FUNCTION_BLOCK CALIBRATE_3P (* 3-point calibration for joysticks (Min, Mid, Max) *)
  (* Standard: 61499-1; Description: Calibrate_3P allows for 3-point calibration of an analog input, ideal for joysticks with center drift. *)
  (* Version 1.0, 2026-05-10, Gemini CLI *)
  PACKAGE OSCAT::Basic::POUs::Engineering::measurements;
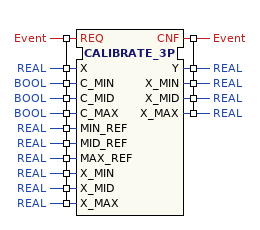
  EVENT_INPUT
    REQ WITH X, C_MIN, C_MID, C_MAX, MIN_REF, MID_REF, MAX_REF, X_MIN, X_MID, X_MAX; (* Normal Execution Request *)
  END_EVENT
  EVENT_OUTPUT
    CNF WITH Y, X_MIN, X_MID, X_MAX; (* Execution Confirmation *)
  END_EVENT
  VAR_INPUT
    X : REAL; (* Raw Input *)
    C_MIN : BOOL; (* Calibrate Min Point *)
    C_MID : BOOL; (* Calibrate Mid Point (Center) *)
    C_MAX : BOOL; (* Calibrate Max Point *)
    MIN_REF : REAL := 0.0; (* Target value for Min *)
    MID_REF : REAL := 50.0; (* Target value for Mid *)
    MAX_REF : REAL := 100.0; (* Target value for Max *)
  END_VAR
  VAR_OUTPUT
    Y : REAL; (* Calibrated Output *)
  END_VAR
  VAR_IN_OUT
    X_MIN : REAL := 0.0; (* Stored Min Value *)
    X_MID : REAL := 50.0; (* Stored Mid Value *)
    X_MAX : REAL := 100.0; (* Stored Max Value *)
  END_VAR
  EC_STATES
    REQ : REQ -> CNF;
  END_STATES
  ALGORITHM REQ IN ST:
(* check for calibration *)
IF C_MIN THEN
	X_MIN := X;
ELSIF C_MID THEN
	X_MID := X;
ELSIF C_MAX THEN
	X_MAX := X;
END_IF;

(* calculate output *)
IF X < X_MID THEN
	IF X_MID > X_MIN THEN
		Y := MIN_REF + (X - X_MIN) * (MID_REF - MIN_REF) / (X_MID - X_MIN);
	ELSE
		Y := MIN_REF;
	END_IF;
ELSE
	IF X_MAX > X_MID THEN
		Y := MID_REF + (X - X_MID) * (MAX_REF - MID_REF) / (X_MAX - X_MID);
	ELSE
		Y := MID_REF;
	END_IF;
END_IF;

(* clipping *)
IF Y < MIN_REF THEN
	Y := MIN_REF;
ELSIF Y > MAX_REF THEN
	Y := MAX_REF;
END_IF;
  END_ALGORITHM
END_FUNCTION_BLOCK
